INTERFACE ITF_PayloadDecoder

END_INTERFACE

(* stored: Version 1.1.0.1
   Itf ITF_PayloadDecoder: Id {9020afa6-913c-4d87-a065-2df612efdf68} *)
